INTERFACE IGear EXTENDS ZApplication.IUnit

PROPERTY PrimaryPositionC : LREAL
GET
END_GET
SET
END_SET
END_PROPERTY

PROPERTY PrimaryVelocityC : LREAL
GET
END_GET
SET
END_SET
END_PROPERTY

END_INTERFACE

(* stored: Version 1.1.0.1
   Itf IGear: Id {80332498-de82-456d-8714-aa13b66ccc93}
   Property PrimaryPositionC: Id {2539f6cb-3b5f-4365-a51d-ce807e3114e5}
   Get Get: Id {6d62e976-34dc-4234-ac52-c30cfe84626b}
   Set Set: Id {ea366428-17b5-469c-91d8-96c6287bd93d}
   Property PrimaryVelocityC: Id {e6a11c7f-4d2e-4461-8251-90942bf8eb6f}
   Get Get: Id {13986ded-ecd3-4267-aea0-64e509bf4c7c}
   Set Set: Id {bfbdd5a4-aa86-4a5f-a77f-677d78b999fe} *)
